PROGRAM P5_03_OtherControl
VAR
END_VAR

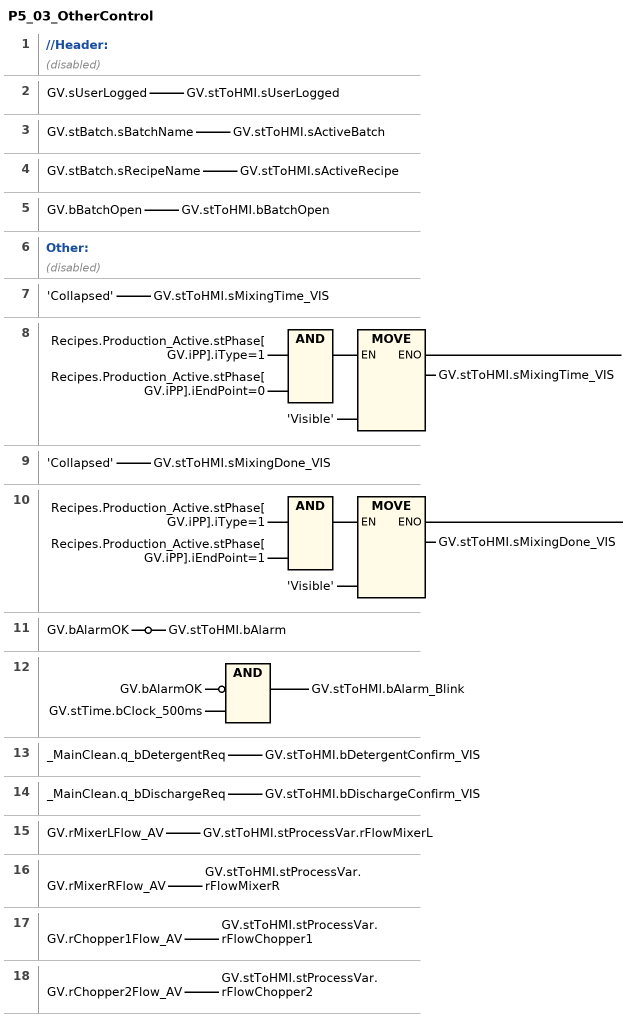
// NETWORK 1 (disabled)
// label: //Header

// NETWORK 2
GV.stToHMI.sUserLogged := GV.sUserLogged;

// NETWORK 3
GV.stToHMI.sActiveBatch := GV.stBatch.sBatchName;

// NETWORK 4
GV.stToHMI.sActiveRecipe := GV.stBatch.sRecipeName;

// NETWORK 5
GV.stToHMI.bBatchOpen := GV.bBatchOpen;

// NETWORK 6 (disabled)
// label: Other

// NETWORK 7
GV.stToHMI.sMixingTime_VIS := 'Collapsed';

// NETWORK 8
IF (Recipes.Production_Active.stPhase[GV.iPP].iType=1) AND (Recipes.Production_Active.stPhase[GV.iPP].iEndPoint=0) THEN
    GV.stToHMI.sMixingTime_VIS := 'Visible';
END_IF

// NETWORK 9
GV.stToHMI.sMixingDone_VIS := 'Collapsed';

// NETWORK 10
IF (Recipes.Production_Active.stPhase[GV.iPP].iType=1) AND (Recipes.Production_Active.stPhase[GV.iPP].iEndPoint=1) THEN
    GV.stToHMI.sMixingDone_VIS := 'Visible';
END_IF

// NETWORK 11
GV.stToHMI.bAlarm := NOT GV.bAlarmOK;

// NETWORK 12
GV.stToHMI.bAlarm_Blink := NOT GV.bAlarmOK AND GV.stTime.bClock_500ms;

// NETWORK 13
GV.stToHMI.bDetergentConfirm_VIS := _MainClean.q_bDetergentReq;

// NETWORK 14
GV.stToHMI.bDischargeConfirm_VIS := _MainClean.q_bDischargeReq;

// NETWORK 15
GV.stToHMI.stProcessVar.rFlowMixerL := GV.rMixerLFlow_AV;

// NETWORK 16
GV.stToHMI.stProcessVar.rFlowMixerR := GV.rMixerRFlow_AV;

// NETWORK 17
GV.stToHMI.stProcessVar.rFlowChopper1 := GV.rChopper1Flow_AV;

// NETWORK 18
GV.stToHMI.stProcessVar.rFlowChopper2 := GV.rChopper2Flow_AV;

END_PROGRAM

(* stored: Version 1.1.0.1
   POU P5_03_OtherControl: Id {3767f6b8-37b7-4d6c-944a-65dae6712b2d}, SpecialFunc None *)
